FUNCTION_BLOCK E_RTimeOut (* Simple implementation of the timeout services *)
  (* Standard: 61499-2; Description: TODO for efficience reasons make this a service interface FB *)
  (* Version 1.0, 2014-10-21, AZ, 4DIAC-Consortium *)
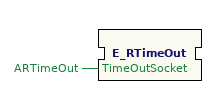
  SOCKETS
    TimeOutSocket : ARTimeOut;
  END_SOCKETS
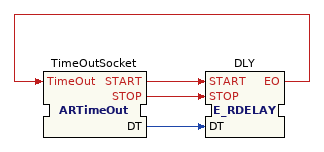
  FBS
    DLY : E_RDELAY;
  END_FBS
  EVENT_CONNECTIONS
    TimeOutSocket.START TO DLY.START;
    TimeOutSocket.STOP TO DLY.STOP;
    DLY.EO TO TimeOutSocket.TimeOut;
  END_CONNECTIONS
  DATA_CONNECTIONS
    TimeOutSocket.DT TO DLY.DT;
  END_CONNECTIONS
END_FUNCTION_BLOCK
